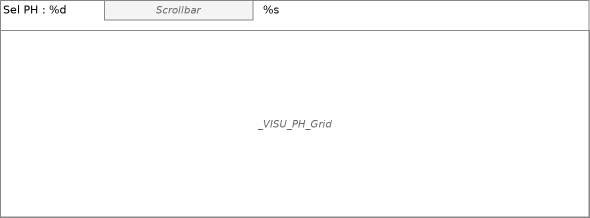
VISUALIZATION VISU_PH_Grid  // 590x218
VAR_IN_OUT
  m_visu_fb : FB_PH_Grid_Visu;       (*visu fb instance*)
END_VAR
    Rectangle (0,0 99x20), "Sel PH : %d", text variable: m_visu_fb.pSelect^
        OnMouseDown: write the text variable via Edit, min m_visu_fb.iBoundLower, max m_visu_fb.iBoundUpper
    Scrollbar (104,0 149x20), tooltip "y-shift"
        p3598130195: m_visu_fb.iBoundLower
        p2245068023: m_visu_fb.iBoundUpper
        p1057716461: m_visu_fb.pSelect^
    Rectangle (260,0 330x20), "%s", text variable: m_visu_fb.pL_Elem_Fb^._pAdsIf^.aO_Name
    Frame (0,30 590x188)
        shows _VISU_PH_Grid(m_Inst := m_visu_fb.pL_Elem_Fb^)
END_VISUALIZATION

(* stored: Version 1.1.0.1, ProductVersion 3.1.4024.3
   Visu VISU_PH_Grid: Id {d1d3cb8e-792f-4cf9-bbe7-264f970b3016} *)
